// TwinCAT 3 PLC project IMAT_Proj
// ProgramVersion: 3.1.4023.0
// libraries:
//   Tc2_Standard, * (Beckhoff Automation GmbH)
//   Tc2_System, * (Beckhoff Automation GmbH)
//   Tc3_Module, * (Beckhoff Automation GmbH)
// project tree:
//   GVLs/ GVL_Safety.TcGVL, KeTop.TcGVL
//   / PlcTask.TcTTO
//   POUs/ MAIN.TcPOU
// real-time tasks:
//   TASK PlcTask: cycle T#10ms, priority 20, ADS port 350
// I/O:
//   DEVICE Device 1 (EtherCAT), AmsNetId 130.246.57.63.2.1
//     Term 1 (EK1200) [EK1200-5000 EtherCAT Power supply (2A E-Bus)]
//       Term 2 (EL6910) [EL6910, TwinSAFE PLC]
//       Term 3 (EL1904) [EL1904, 4 Ch. Safety Input 24V, TwinSAFE]
//         modules: Module 1 (FSOES)
//       Term 4 (EL2904) [EL2904, 4 Ch. Safety Output 24V, 0.5A, TwinSAFE]
//         modules: Module 1 (FSOES), Module 2 (DO)
//       Term 5 (EL1904) [EL1904, 4 Ch. Safety Input 24V, TwinSAFE]
//         modules: Module 1 (FSOES)
//       Term 6 (EL1904) [EL1904, 4 Ch. Safety Input 24V, TwinSAFE]
//         modules: Module 1 (FSOES)
//       Term 14 (EL1904) [EL1904, 4 Ch. Safety Input 24V, TwinSAFE]
//         modules: Module 1 (FSOES)
//       Term 7 (EK1110)
// variable links:
//   (this object) <-> Device 1 (EtherCAT)/Term 1 (EK1200)/Term 14 (EL1904)
//     Term 1 (EK1200)/Term 2 (EL6910)/ConnectionInputs/Message_15 TxPDO <-> Module 1 (FSOES)/RxPDO/FSOE
//     Term 1 (EK1200)/Term 2 (EL6910)/ConnectionOutputs/Message_15 RxPDO <-> Module 1 (FSOES)/TxPDO/FSOE
//   (this object) <-> Device 1 (EtherCAT)/Term 1 (EK1200)/Term 2 (EL6910)
//     Term 1 (EK1200)/Term 14 (EL1904)/Module 1 (FSOES)/RxPDO/FSOE <-> ConnectionInputs/Message_15 TxPDO
//     Term 1 (EK1200)/Term 3 (EL1904)/Module 1 (FSOES)/RxPDO/FSOE <-> ConnectionInputs/Message_2 TxPDO
//     Term 1 (EK1200)/Term 4 (EL2904)/Module 1 (FSOES)/RxPDO/FSOE <-> ConnectionInputs/Message_3 TxPDO
//     Term 1 (EK1200)/Term 5 (EL1904)/Module 1 (FSOES)/RxPDO/FSOE <-> ConnectionInputs/Message_6 TxPDO
//     Term 1 (EK1200)/Term 6 (EL1904)/Module 1 (FSOES)/RxPDO/FSOE <-> ConnectionInputs/Message_9 TxPDO
//     Term 1 (EK1200)/Term 14 (EL1904)/Module 1 (FSOES)/TxPDO/FSOE <-> ConnectionOutputs/Message_15 RxPDO
//     Term 1 (EK1200)/Term 3 (EL1904)/Module 1 (FSOES)/TxPDO/FSOE <-> ConnectionOutputs/Message_2 RxPDO
//     Term 1 (EK1200)/Term 4 (EL2904)/Module 1 (FSOES)/TxPDO/FSOE <-> ConnectionOutputs/Message_3 RxPDO
//     Term 1 (EK1200)/Term 5 (EL1904)/Module 1 (FSOES)/TxPDO/FSOE <-> ConnectionOutputs/Message_6 RxPDO
//     Term 1 (EK1200)/Term 6 (EL1904)/Module 1 (FSOES)/TxPDO/FSOE <-> ConnectionOutputs/Message_9 RxPDO
//   (this object) <-> Device 1 (EtherCAT)/Term 1 (EK1200)/Term 3 (EL1904)
//     Term 1 (EK1200)/Term 2 (EL6910)/ConnectionInputs/Message_2 TxPDO <-> Module 1 (FSOES)/RxPDO/FSOE
//     Term 1 (EK1200)/Term 2 (EL6910)/ConnectionOutputs/Message_2 RxPDO <-> Module 1 (FSOES)/TxPDO/FSOE
//   (this object) <-> Device 1 (EtherCAT)/Term 1 (EK1200)/Term 4 (EL2904)
//     Term 1 (EK1200)/Term 2 (EL6910)/ConnectionInputs/Message_3 TxPDO <-> Module 1 (FSOES)/RxPDO/FSOE
//     Term 1 (EK1200)/Term 2 (EL6910)/ConnectionOutputs/Message_3 RxPDO <-> Module 1 (FSOES)/TxPDO/FSOE
//   (this object) <-> Device 1 (EtherCAT)/Term 1 (EK1200)/Term 5 (EL1904)
//     Term 1 (EK1200)/Term 2 (EL6910)/ConnectionInputs/Message_6 TxPDO <-> Module 1 (FSOES)/RxPDO/FSOE
//     Term 1 (EK1200)/Term 2 (EL6910)/ConnectionOutputs/Message_6 RxPDO <-> Module 1 (FSOES)/TxPDO/FSOE
//   (this object) <-> Device 1 (EtherCAT)/Term 1 (EK1200)/Term 6 (EL1904)
//     Term 1 (EK1200)/Term 2 (EL6910)/ConnectionInputs/Message_9 TxPDO <-> Module 1 (FSOES)/RxPDO/FSOE
//     Term 1 (EK1200)/Term 2 (EL6910)/ConnectionOutputs/Message_9 RxPDO <-> Module 1 (FSOES)/TxPDO/FSOE
//   IMAT_Proj Instance <-> Device 1 (EtherCAT)/Term 1 (EK1200)/Term 2 (EL6910)
//     PlcTask Inputs/GVL_Safety.NORMALMODE_FB_STATE <-> Function Block Info Data/TwinSafeGroup1.Network3_OPMODE.FBAnd1 Info Data/State
//     PlcTask Outputs/GVL_Safety.ERRACK <-> StandardOutputs/Standard In Var 1
//     PlcTask Outputs/GVL_Safety.MUTE_ENABLING <-> StandardOutputs/Standard In Var 18
//     PlcTask Outputs/GVL_Safety.MUTE_LC <-> StandardOutputs/Standard In Var 17
//     PlcTask Outputs/GVL_Safety.SAFETYRUN <-> StandardOutputs/Standard In Var 4

CONFIGURATION IMAT_Proj
    RESOURCE PLC ON TwinCAT3
        TASK PlcTask(INTERVAL := T#10ms, PRIORITY := 20);
        PROGRAM MAIN WITH PlcTask : MAIN;
    END_RESOURCE
END_CONFIGURATION

// ---- GVLs/GVL_Safety.TcGVL
{attribute 'qualified_only'}
VAR_GLOBAL
    
    SAFETYRUN AT %Q* : BOOL := TRUE;
    ERRACK AT %Q* : BOOL;
    MUTE_LC AT %Q* : BOOL := FALSE;
    MUTE_ENABLING AT %Q* : BOOL := FALSE;
    UNMUTE_ENABLING AT %Q* : BOOL;
    NORMALMODE_FB_STATE AT %I*: USINT;
END_VAR

// ---- GVLs/KeTop.TcGVL
{attribute 'qualified_only'}
VAR_GLOBAL
    alive : UINT;
    keys: ARRAY[0..127] OF BOOL;
    buzzer : UINT;
    keySwitch : BYTE;
    enSwitch : BYTE;
END_VAR

// ---- POUs/MAIN.TcPOU
PROGRAM MAIN
VAR
    
END_VAR

END_PROGRAM
